(*
Logs a debug message as a string without associating it with a specific component.
*)
FUNCTION DebugStr
VAR_INPUT
	sInfo			: Str;
END_VAR
VAR
END_VAR

IF _Debug.nLastStr < Param.DEBUGSTR_CAP THEN
	_Debug.nLastStr := _Debug.nLastStr + 1;
ELSE
	_Debug.nLastStr := 1;
END_IF

_Debug.debugStr[_Debug.nLastStr] := sInfo;

END_FUNCTION

(* stored: Version 1.1.0.1
   POU DebugStr: Id {34717bf4-9bf9-4a89-a482-5331f33a4582}, SpecialFunc None *)
